{attribute addProperty BoxType "EL3124-0000-0016"}
{attribute addProperty Id "AI_Standard_ChannelAT %I*ARRAY[0..3] OF AI_Standard_Channel_904746A2128160WcStateAT %I*WcState_98A4DF7520.250InfoDataAT %I*InfoData_BC63D37F80100"}
{attribute addProperty CRC "1712706657"}
{attribute addProperty SizeInBites "210"}
{attribute addProperty SizeInBytes "26.25"}
TYPE EL3124_6082EBFD :
STRUCT
	{attribute addProperty Name "AI_Standard_Channel"}
	AI_Standard_Channel : ARRAY[0..3] OF AI_Standard_Channel_904746A2;
	{attribute addProperty Name "WcState"}
	WcState : WcState_98A4DF75;
	{attribute addProperty Name "InfoData"}
	InfoData : InfoData_BC63D37F;
END_STRUCT
END_TYPE

(* stored: Version 1.2.0.0, ProductVersion 3.1.4024.9
   DUT EL3124_6082EBFD: Id {5b638750-f8dc-4a97-a52a-769bcde6b5f0} *)
